            (* split slave state and link state *)
            FOR I := 0 TO MIN(iNumOfSlavesRead, iSLAVEADDR_ARR_SIZE) DO
                (* slave state*)
                arrSlaveInfo[I].stState.eEcState 		:= arrSlaveStates[I].deviceState AND 16#0F;
                arrSlaveInfo[I].stState.bError 			:= arrSlaveStates[I].deviceState.4;
                arrSlaveInfo[I].stState.bInvalidVPRS 	:= arrSlaveStates[I].deviceState.5;
                (* link state *)
                arrSlaveInfo[I].stState.bNoCommToSlave 	:= arrSlaveStates[I].linkState.0;
                arrSlaveInfo[I].stState.bLinkError 		:= arrSlaveStates[I].linkState.1;
                arrSlaveInfo[I].stState.bMissingLink 	:= arrSlaveStates[I].linkState.2;
                arrSlaveInfo[I].stState.bUnexpectedLink := arrSlaveStates[I].linkState.3;
                arrSlaveInfo[I].stState.bPortA 			:= arrSlaveStates[I].linkState.4;
                arrSlaveInfo[I].stState.bPortB 			:= arrSlaveStates[I].linkState.5;
                arrSlaveInfo[I].stState.bPortC 			:= arrSlaveStates[I].linkState.6;
                arrSlaveInfo[I].stState.bPortD 			:= arrSlaveStates[I].linkState.7;
                (* DiagData *)
                arrSlaveInfo[I].bDiagData	:= ((arrSlaveStates[I].deviceState AND 16#F0) <> 0) OR
                    (((arrSlaveStates[I].deviceState AND 16#0F) > 0) AND ((arrSlaveStates[I].deviceState AND 16#0F) < 8)) OR
                    (arrSlaveStates[I].linkState <> 0);

                IF arrSlaveInfo[I].bDiagData THEN
                    IF (I=0) THEN
                        aiDiagIndex[0] := 0;
                    ELSE
                        IF (aiDiagIndex[0] = 0) AND NOT arrSlaveInfo[0].bDiagData THEN
                            aiDiagIndex[0] :=  UDINT_TO_UINT(I);
                        END_IF
                    END_IF
                END_IF
            END_FOR
        END_IF
    END_IF

    IF arrSlaveInfo[aiDiagIndex[0]].bDiagData THEN
        iState := E_EcatDiagState.GetTopoDataLen;
    ELSE
        FOR I := 0 TO ESC_MAX_PORTS DO
            MEMSET(ADR(arrDiagSlaveInfo[I]), 0, SIZEOF(arrDiagSlaveInfo[I]));
            MEMSET(ADR(arrDiagSlaveInfoScanned[I]), 0, SIZEOF(arrDiagSlaveInfoScanned[I]));
        END_FOR
        iState := E_EcatDiagState.Done;
    END_IF
END_IF
END_ACTION

ACTION M_GetTopoData:
fbGetTopologyData(
    NETID	:= sMasterNetID,
    PORT	:= 16#FFFF,
    IDXGRP	:= 16#22,
    IDXOFFS	:= 0,
    LEN		:= iTopologyData*SIZEOF(arrTopologyData[0]),
    DESTADDR:= ADR(arrTopologyData),
    READ	:= TRUE,
    TMOUT	:= tTimeout,
);

IF NOT fbGetTopologyData.BUSY THEN
    fbGetTopologyData(READ := FALSE);

    IF NOT fbGetTopologyData.ERR THEN
        aiDiagPort[0] := arrTopologyData[aiDiagIndex[0]].iOwnPhysicalAddr;
        aiDiagPort[1] := arrTopologyData[aiDiagIndex[0]].stPhysicalAddr.portB;
        aiDiagPort[2] := arrTopologyData[aiDiagIndex[0]].stPhysicalAddr.portC;
        aiDiagPort[ESC_MAX_PORTS] := arrTopologyData[aiDiagIndex[0]].stPhysicalAddr.portD;

        (* clear diag index  *)
        aiDiagIndex[1] := 0;
        aiDiagIndex[2] := 0;
        aiDiagIndex[ESC_MAX_PORTS] := 0;

        (* find slaves on PortB-D of first slave with diag *)
        FOR P := 0 TO ESC_MAX_PORTS DO
            IF aiDiagPort[P] <> 0 THEN
            FOR I := 0 TO MIN(iTopologyData-1,iSLAVEADDR_ARR_SIZE) DO
                IF arrTopologyData[I].iOwnPhysicalAddr = aiDiagPort[P] THEN
                    aiDiagIndex[P] := UDINT_TO_UINT(I);
                    EXIT;
                END_IF
            END_FOR
        END_IF
        END_FOR
    END_IF

    iIdx := 0;
    iState := E_EcatDiagState.ScanSlaves;
END_IF
END_ACTION

ACTION M_GetTopoDataLen:
fbGetTopologyData(
    NETID	:= sMasterNetID,
    PORT	:= 16#FFFF,
    IDXGRP	:= EC_ADS_IGRP_MASTER_COUNT_SLAVE,
    IDXOFFS	:= EC_ADS_IOFFS_MASTER_COUNT_SLAVE,
    LEN		:= SIZEOF(iTopologyData),
    DESTADDR:= ADR(iTopologyData),
    READ	:= TRUE,
    TMOUT	:= tTimeout,
);

IF NOT fbGetTopologyData.BUSY THEN
    fbGetTopologyData(READ := FALSE);

    iState := E_EcatDiagState.GetTopoData;
END_IF
END_ACTION

ACTION M_ScanSlaves:
fbEcGetScannedSlaves(
    bExecute				:= TRUE,
    sNetId					:= sMasterNetID,
    pArrEcScannedSlaveInfo	:= ADR(arrScannedSlaveInfo),
    cbBufLen				:= SIZEOF(arrScannedSlaveInfo),
    tTimeout				:= tTimeout
);

IF NOT fbEcGetScannedSlaves.bBusy THEN
    fbEcGetScannedSlaves(bExecute := FALSE);

    IF fbEcGetScannedSlaves.bError THEN
        nScannedSlaves := 0;
    ELSE
        nScannedSlaves := fbEcGetScannedSlaves.nSlaves;
    END_IF

    iState := E_EcatDiagState.GetSlaveIdentity;

END_IF
END_ACTION

END_FUNCTION_BLOCK

// ---- POUs/Functions/FB_EcatDiag.TcPOU
(*
Ecat bus diagnostic tool
2015-11-4 Alex Wallace
This function block checks the states of all slaves on the ecat bus network,
it could be modified to export the states of the slaves on an individual basis,
but for now it sets the output boolean true if all slaves are OP and false otherwise.
To start the block provide a falling edge on the first pass boolean input.

2018-05-05 Margaret Ghaly
Function block has been modified to retrieve the Device State of the Ethercat Master.
It also exports the states and information of each individual configured Slave.
And saves them in the array q_aEcConfSlaveInfo.
*)
FUNCTION_BLOCK FB_EcatDiag
VAR_INPUT
    {attribute 'naming' := 'omit'}
    I_AMSNetId AT %I* : AMSNETID; //Link to the AMSNETID name in the ethercat master info.
    i_xFirstPass: BOOL; //Hook to system first pass boolean for proper intialization (must be true for the first cycle of the PLC)
END_VAR
VAR_OUTPUT
    q_xAllSlaveStatesGood: BOOL; // Set to True if all Slaves are in OP State
    q_anTermStates: ARRAY[1..256] OF BYTE; //ECAT State of terminals in the bus
    q_xMasterStateGood:BOOL; // Set to True if the Master Device State is OP
    q_nMasterState: WORD; // The Device State of the Master
    q_sMasterState:STRING; //State of the ECAT master
    q_astEcConfSlaveInfo :  ARRAY[1..256] OF ST_EcDevice; //State of all ECAT slaves in the bus
    q_nSlaves: UINT; // the Number of the connected Slaves
END_VAR
VAR
    sNetId: T_AmsNetId; //NetId string
    astTermStates: ARRAY[1..256] OF ST_EcSlaveState; //ECAT Slave States Buffer
    astEcConfSlaveInfo: ARRAY[1..256] OF ST_EcSlaveConfigData; //ECAT Slave Configs Buffer
    fbGetAllSlaveStates: FB_EcGetAllSlaveStates; //Acquires the ECAT Slave States puts them into astTermStates

    fbGetMasterState: FB_EcGetMasterState; //Acquires ECAT Master State
    fbGetConfSlaves: FB_EcGetConfSlaves; //Acquires the ECAT slave configuration of the bus (how many, what kind, etc)
    {attribute 'naming' := 'omit'}
    ftReset: F_TRIG; //Reset trigger sensor
    {attribute 'naming' := 'omit'}
    ftMasterReset: F_TRIG; //Retrigger sensor for GetMasterState
    nIterator: INT; //Generic iterator placeholder
END_VAR

//Create the net ID string
sNetId := F_CreateAmsNetId(I_AMSNetId);

//Query the state of all terminals, collect in astTermStates
ftReset(CLK:=fbGetAllSlaveStates.bBusy OR i_xFirstPass);
fbGetAllSlaveStates.bExecute := ftReset.Q;
fbGetAllSlaveStates(sNetId:=sNetId, pStateBuf := ADR(astTermStates), cbBufLen:=SIZEOF(astTermStates));
//Keep checking...



//Cycle through each entry in the array and check if we have anyone not in OP and that the link state is good.
// If so, then set our global IO bad boolean.
IF fbGetAllSlaveStates.nSlaves > 0 THEN
    q_xAllSlaveStatesGood := TRUE;
FOR nIterator := 1 TO (UINT_TO_INT(fbGetAllSlaveStates.nSlaves) ) BY 1
    DO
    IF NOT( (astTermStates[nIterator].deviceState = EC_DEVICE_STATE_OP) AND (astTermStates[nIterator].linkState = EC_LINK_STATE_OK)) THEN
        q_xAllSlaveStatesGood := FALSE;
    END_IF
    q_anTermStates[nIterator] := astTermStates[nIterator].deviceState;
    q_astEcConfSlaveInfo[nIterator].nDeviceState :=astTermStates[nIterator].deviceState;//
    q_astEcConfSlaveInfo[nIterator].nLinkState :=astTermStates[nIterator].linkState;//
    q_astEcConfSlaveInfo[nIterator].sDeviceState:= F_ConvSlaveStateToString(state:=astTermStates[nIterator]);//

END_FOR
END_IF

// Read the EtherCAT state of the master. If the call is successful,
//the State output variable of type WORD contains the requested status information.
ftMasterReset(CLK:=fbGetMasterState.bBusy OR i_xFirstPass);
fbGetMasterState(sNetId:= sNetId, bExecute:=ftMasterReset.Q,
                state => q_nMasterState,bError=>,
                nErrId=>);
q_xMasterStateGood:= (fbGetMasterState.state = BYTE_TO_UINT(EC_DEVICE_STATE_OP));
q_sMasterState := F_ConvMasterDevStateToString(fbGetMasterState.state);

//This function is used to read a list of all configured slaves from the EtherCat master object Directory
//needs to run only once
fbGetConfSlaves(bExecute := i_xFirstPass, sNetId :=sNetId, pArrEcConfSlaveInfo := ADR(astEcConfSlaveInfo),cbBufLen := SIZEOF(astEcConfSlaveInfo));
q_nSlaves:=fbGetConfSlaves.nSlaves;

IF  NOT (fbGetConfSlaves.bBusy) THEN
    FOR nIterator := 1 TO (UINT_TO_INT(fbGetConfSlaves.nSlaves) ) BY 1
    DO
    q_astEcConfSlaveInfo[nIterator].nAddrr :=astEcConfSlaveInfo[nIterator].nAddr;
    q_astEcConfSlaveInfo[nIterator].sName :=astEcConfSlaveInfo[nIterator].sName;
    q_astEcConfSlaveInfo[nIterator].sType :=astEcConfSlaveInfo[nIterator].sType;
END_FOR
    fbGetConfSlaves.bExecute := FALSE;
END_IF

END_FUNCTION_BLOCK

// ---- POUs/Functions/FB_Index.TcPOU
(* Index FB
A. Wallace 2016-9-3

Why doesn't beckhoff have this as a builtin type?

Use this thing to have a simple indexer with rollover.

*)
FUNCTION_BLOCK FB_Index
VAR_INPUT
    {attribute 'naming' := 'off'}
    LowerLimit : INT := 1; //Incrementer will rollver over to this value (and initialize to this value)
    ValInc : INT := 1; //Incrementer increments by this value
    UpperLimit	:	INT := 1; //Incrementer will rollover at this value to lower limit
    {attribute 'naming' := 'off'}
END_VAR
VAR_OUTPUT

END_VAR
VAR
    nVal	:	INT := LowerLimit; //Internal incrementer value, initialized to LowerLimit
END_VAR

{analysis -2} //Only the methods and actions are needed

ACTION Dec:
nVal := nVal - ValInc;
IF nVal < LowerLimit THEN nVal := UpperLimit; END_IF
END_ACTION

//Decrement the counter and return new value
METHOD DecVal : INT
VAR_INPUT
END_VAR
Dec();
DecVal := nVal;
END_METHOD

ACTION Inc:
// Dont use this, use ValInc
nVal := nVal + ValInc;
IF nVal >  UpperLimit THEN nVal := LowerLimit; END_IF
END_ACTION

//Increment the counter and return new value
METHOD PUBLIC IncVal : INT
VAR_INPUT
END_VAR
Inc();
IncVal := nVal;
END_METHOD

END_FUNCTION_BLOCK

// ---- POUs/Functions/FB_UnixTimeStampGlobal.TcPOU
FUNCTION_BLOCK FB_UnixTimeStampGlobal
(*
    Runs FB_UnixTimeStamp and stuffs the result into this library's GVL
    2019-10-09 Zachary Lentz
*)
VAR_INPUT
    // If TRUE, we will update the output on this cycle.
    bExecute: BOOL;
END_VAR
VAR_OUTPUT
END_VAR
VAR
    fbTimeStamp: FB_UnixTimeStamp;
END_VAR

fbTimeStamp(
    bExecute := bExecute,
    fTime => DefaultGlobals.fTimeStamp);

END_FUNCTION_BLOCK

// ---- POUs/Functions/FB_XKoyoPLCModbus.TcPOU
//Facilitates communication between Beckhoff and Koyo PLC over the network.
FUNCTION_BLOCK FB_XKoyoPLCModbus
VAR
    fbKoyo_PLCInputCoilsRx	:	FB_MBReadCoils; //FB for reading the coils from the other PLC
    anKoyo_PLC_CnBits	:	ARRAY [0..20] OF BYTE; //Buffer for coil readbacks
    {attribute 'naming' := 'omit'}
    ftReset	: F_TRIG; //Reset edge sensor
    {attribute 'naming' := 'omit'}
    tonRetry : TON; //Retry timer
    nIndex : INT; //Index for clearing the coil array
END_VAR

VAR_INPUT
    i_tRetryTime : TIME := T#10S; //Retry time if modbus transaction fails
    i_sIPAddr	 : STRING[15]; //IP address of the Koyo PLC
END_VAR

VAR_OUTPUT
    q_xNoPLCResponse : BOOL := TRUE; //Could not reach the PLC if true
    q_anPLCResponse   : ARRAY [0..20] OF BYTE; //Buffer of coils retrieved from the other PLC
    q_xError         : BOOL := FALSE; //Transaction or other error
END_VAR

(* Look ma' no wires! *)
(* A. Wallace, 2015-7-22
XKoyoPLCModbus

Facilitates communication between Beckhoff and Koyo PLC over the network.

Useful if you don't have time to run a wire. Fairly reliable.

*)

(* Modbus Info for Koyo
Modbus Addresses for
Koyo DL05/06/240/250/260/430/440/450 PLCs
PLC Memory Type		| Modbus start address Decimal (octal) | Function codes
Inputs (X)			  2048 (04000)							2
Special Relays (SP)	  3072 (06000)							2
Outputs (Y)			  2048 (04000)							1, 5, 15
Control Relays (C)	  3072 (06000)							1, 5, 15
Timer Contacts (T)	  6144 (014000)							1, 5, 15
Counter Contacts (CT) 6400 (014400)							1, 5, 15
Stage Status Bits (S) 6144 (012000)							1, 5, 15
*)

(* Begin code *)
// Retry after some time
tonRetry.IN := NOT fbKoyo_PLCInputCoilsRx.bBusy;
tonRetry.PT := i_tRetryTime;
tonRetry();

ftReset(CLK:=fbKoyo_PLCInputCoilsRx.bBusy);
ftReset();

fbKoyo_PLCInputCoilsRx.bExecute := ftReset.Q OR tonRetry.Q;

fbKoyo_PLCInputCoilsRx(sIPAddr:='i_sIPAddr', nTCPPort:=502, nQuantity:=32, nMBAddr:=8#6000, cbLength:=USINT_TO_UDINT(SIZEOF(anKoyo_PLC_CnBits)),  pDestAddr:=ADR(anKoyo_PLC_CnBits), tTimeout:=T#10S);

//run some error code for modbus
IF fbKoyo_PLCInputCoilsRx.bError THEN
    //if there's a modbus error, set all incoming bits to zero
    {analysis -41} //There are one-liners for resetting an array to zero but they don't comply with 61131
    FOR nIndex := 0 TO USINT_TO_INT(SIZEOF(anKoyo_PLC_CnBits))-1 DO //starts at 0
        anKoyo_PLC_CnBits[nIndex]:=0;
    END_FOR
    {analysis +41}
    q_xError := TRUE;

ELSIF ftReset.Q AND fbKoyo_PLCInputCoilsRx.cbRead > 0 THEN
    fbKoyo_PLCInputCoilsRx.bExecute := FALSE;
    q_xNoPLCResponse:= FALSE;
    q_xError := FALSE;

//more error code cause we didn't manage to read anything
ELSIF fbKoyo_PLCInputCoilsRx.cbRead = 0 THEN
    q_xError := TRUE;
    q_xNoPLCResponse:= TRUE;

END_IF

q_anPLCResponse := anKoyo_PLC_CnBits;

END_FUNCTION_BLOCK

// ---- POUs/Hardware/FB_AnalogOutput.TcPOU
FUNCTION_BLOCK FB_AnalogOutput
(*
    Converts a real unit value (e.g., volts) to the integer needed for an analog output terminal.
    2019-10-09 Zachary Lentz
*)
VAR_INPUT
    // The real value to send to the output
    fReal: LREAL;
    // The maximum allowed real value for the connected hardware
    fSafeMax: LREAL;
    // The minimum allowed real value for the connected hardware
    fSafeMin: LREAL;
    // The number of bits correlated with the terminal's max output. This is not necessarily the resolution parameter.
    iTermBits: UINT;
    // The fReal value correlated with the terminal's max output
    fTermMax: LREAL;
    // The fReal value correlated with the terminal's min output
    fTermMin: LREAL;
END_VAR
VAR_OUTPUT
    // Connect this output to the terminal
    iRaw AT %Q*: INT;
END_VAR
VAR
    fScale: LREAL;
END_VAR

// Set the scaling from real to raw
IF fScale = 0 AND fTermMax > fTermMin THEN
    fScale := (EXPT(2, iTermBits) - 1) / (fTermMax - fTermMin);
END_IF

// Adjust real value to be within the limits
fReal := MIN(fReal, fSafeMax, fTermMax);
fReal := MAX(fReal, fSafeMin, fTermMin);

// Scale the output accordingly
iRaw := LREAL_TO_INT((fReal - fTermMin) * fScale);

END_FUNCTION_BLOCK

// ---- POUs/Hardware/FB_AnalogInput.TcPOU
FUNCTION_BLOCK FB_AnalogInput
(*
    Converts the integer from an analog input terminal to a real unit value (e.g., volts)
    2019-10-09 Zachary Lentz
*)
VAR_INPUT
    // Connect this input to the terminal
    iRaw AT %I*: INT;
    // The number of bits correlated with the terminal's max value. This is not necessarily the resolution parameter.
    iTermBits: UINT;
    // The fReal value correlated with the terminal's max value
    fTermMax: LREAL;
    // The fReal value correlated with the terminal's min value
    fTermMin: LREAL;
END_VAR
VAR_OUTPUT
    // The real value read from the output
    fReal: LREAL;
END_VAR
VAR
    fScale: LREAL;
END_VAR

IF fScale = 0 AND fTermMax > fTermMin THEN
    fScale := (EXPT(2, iTermBits) - 1) / (fTermMax - fTermMin);
END_IF
IF fScale <> 0 THEN
    fReal := iRaw / fScale + fTermMin;
END_IF

END_FUNCTION_BLOCK

// ---- POUs/Hardware/FB_CoE_FastRead.TcPOU
FUNCTION_BLOCK FB_CoE_FastRead
(*
    Utility to repeatedly read a CoE parameter
    2019-10-09 Zachary Lentz

    In practice, it's impossible to read most CoE parameters every cycle,
    but this is a best effort and will work if the data is available
*)
VAR_INPUT
    // If TRUE we'll attempt a CoE read this cycle.
    bExecute: BOOL;
    // Link this to your terminal's drive reference variables under InfoData.
    stPlcDriveRef AT %I*: ST_PlcDriveRef;
    // Hexadecimal index of CoE, e.g. the 8010 in 8010:12
    nIndex: UINT;
    // Hexadecimal subindex of CoE, e.g. the 12 in 8010:12
    nSubIndex: BYTE;
    // Pointer to a value to fill with the result of the read, e.g. ADR(MyValue)
    pDstBuf: PVOID;
    // Data size of pDstBuf, e.g. SIZEOF(MyValue)
    cbBufLen: UINT;
END_VAR
VAR_OUTPUT
    // TRUE if the value was updated on this cycle.
    bNewValue: BOOL;
END_VAR
VAR
    fbRead: FB_CoERead_ByDriveRef;
    stDriveRef: ST_DriveRef;
    iLoop: INT;
    bInnerExec: BOOL;
END_VAR

stDriveRef.sNetId := F_CreateAmsNetId(stPlcDriveRef.aNetId);
stDriveRef.nSlaveAddr := stPlcDriveRef.nSlaveAddr;
stDriveRef.nDriveNo := stPlcDriveRef.nDriveNo;
stDriveRef.nDriveType := stPlcDriveRef.nDriveType;

bNewValue := FALSE;
IF bExecute THEN
    // You need to do this block 3 times per cycle to have a chance at always getting a read
    FOR iLoop:= 1 TO 3 DO
        fbRead(
            stDriveRef := stDriveRef,
            nIndex := nIndex,
            nSubIndex := nSubIndex,
            pDstBuf := pDstBuf,
            cbBufLen := cbBufLen,
            bExecute := bInnerExec,
            tTimeout := T#1s);

        IF bInnerExec AND NOT fbRead.bBusy AND NOT fbRead.bError THEN
            bInnerExec := FALSE;
            bNewValue := TRUE;
        ELSE
            bInnerExec := TRUE;
        END_IF
    END_FOR
END_IF

END_FUNCTION_BLOCK

// ---- POUs/Hardware/FB_EL6_Com.TcPOU
FUNCTION_BLOCK FB_EL6_Com
(*
    Communicate with a serial device connected to an EL6XXX
    2019-10-09 Zachary Lentz and Jackson Sheppard

    May contain assumptions about the device we wrote it for, potentially will need to be adjusted
*)
VAR_INPUT
    // Command to send to the serial device
    {attribute 'pytmc' := '
        pv: CMD
        io: io
    '}
    sCmd: STRING;

    // Pulse this to TRUE and back to FALSE when it's time to send
    {attribute 'pytmc' := '
        pv: SEND
        io: io
    '}
    bSend: BOOL;

    // Any static prefix to add before every sent message
    sSendPrefix: STRING;
    // Any static suffix to add after every sent message
    sSendSuffix: STRING;
    // Any static prefix to strip off of every recieved message
    sRecvPrefix: STRING;
    // Any static suffic to strip off of every recieved message
    sRecvSuffix: STRING;
    tTimeout: TIME := T#1S;
END_VAR
VAR_IN_OUT
    stIn_EL6: EL6inData22B;
    stOut_EL6: EL6outData22B;
END_VAR
VAR_OUTPUT
    // The response recieved from the serial device
    {attribute 'pytmc' := '
        pv: RESP
        io: input
    '}
    sResponse: STRING;

    // This is set to TRUE after recieving a response
    {attribute 'pytmc' := '
        pv: DONE
        io: input
    '}
    bDone: BOOL;

    {attribute 'pytmc' := '
        pv: ERR:SER
        io: input
    '}
    eSerialLineErrorID: ComError_t;

    {attribute 'pytmc' := '
        pv: ERR:SEND
        io: input
    '}
    eSendErrorID: ComError_t;

    {attribute 'pytmc' := '
        pv: ERR:RECV
        io: input
    '}
    eRecvErrorID: ComError_t;
END_VAR
VAR
    // Communication Buffers
    TxBuffer: ComBuffer;
    RxBuffer: ComBuffer;
    fbClearComBuffer: ClearComBuffer;

    // Parameters for PLC -> EL6
    fbEL6Ctrl: SerialLineControl;
    bEL6CtrlError: BOOL;
    eEL6CtrlErrorID: ComError_t;

    // Parameters for EL6 -> Serial Device
    fbSend: SendString;
    bSendBusy: BOOL;
    eLastSendErrorID: ComError_t;
    fbReceive: ReceiveString;
    sReceivedString: STRING;
    sLastReceivedString: STRING;
    bStringReceived: BOOL;
    bReceiveBusy: BOOL;
    bReceiveError: BOOL;
    eReceiveErrorID: ComError_t;
    bReceiveTimeout: BOOL;
    nReceiveCounter: UDINT;
    nSendCounter: UDINT;
    sStringToSend: STRING;
    fbFormatString: FB_FormatString;

    // Parameters for state-machine implementation
    nStep: INT := 0;
END_VAR

fbEL6Ctrl(
    Mode:= SERIALLINEMODE_EL6_22B,
    pComIn:= ADR(stIn_EL6),
    pComOut:= ADR(stOut_EL6),
    SizeComIn:= UINT_TO_INT(SIZEOF(stIn_EL6)),
    Error=> ,
    ErrorID=> eSerialLineErrorID,
    TxBuffer:= TxBuffer,
    RxBuffer:= RxBuffer );
IF fbEL6Ctrl.Error THEN
    bEL6CtrlError := TRUE;
    eEL6CtrlErrorID := fbEL6Ctrl.ErrorID;
END_IF
IF bSend THEN
    nStep := 10;
    bSend := FALSE;
    bDone := FALSE;
END_IF
// Attempt at solution that sends one command at a time, not on constant loop
CASE nStep OF
    0:
        ; // idle
    10:
        // Clear buffers in case any lingering data
        fbClearComBuffer(Buffer:=TxBuffer);
        fbClearComBuffer(Buffer:=RxBuffer);
        // Prepare string to send
        sStringToSend := CONCAT(sSendPrefix, CONCAT(sCmd, sSendSuffix));
        // Send string
        fbSend(	SendString:= sStringToSend,
                TXbuffer:= TxBuffer,
                Busy=> bSendBusy,
                Error=> eSendErrorID);
        IF fbSend.Error <> COMERROR_NOERROR THEN
            eLastSendErrorID := fbSend.Error;
        ELSE
            nSendCounter := nSendCounter + 1;
        END_IF
        nStep := nStep + 10;
    20:
        // Finish sending String
        IF fbSend.Busy THEN
            fbSend(	SendString:= sStringToSend,
                    TXbuffer:= TxBuffer,
                    Busy=> bSendBusy,
                    Error=> eSendErrorID);
            IF fbSend.Error <> COMERROR_NOERROR THEN
                eLastSendErrorID := fbSend.Error;
            ELSE
                nSendCounter := nSendCounter + 1;
            END_IF
        ELSE
            nStep := nStep + 10;
        END_IF
    30:
        // Get Reply
        fbReceive(
            Prefix:= sRecvPrefix,
            Suffix:= sRecvSuffix,
            Timeout:= tTimeout,
            ReceivedString:= sReceivedString,
            RXbuffer:= RxBuffer,
            StringReceived=> bStringReceived,
            Busy=> bReceiveBusy,
            Error=> eRecvErrorID,
            RxTimeout=> bReceiveTimeout );
        IF fbReceive.Error <> COMERROR_NOERROR THEN
            eReceiveErrorID := fbReceive.Error;
        END_IF
        IF bStringReceived THEN
            nReceiveCounter := nReceiveCounter + 1;
            // Check for response
            IF FIND(sReceivedString, sStringToSend)=0 THEN
                sResponse := sReceivedString;
                bDone := TRUE;
                nStep := 0;
            END_IF
        END_IF
END_CASE

END_FUNCTION_BLOCK

// ---- POUs/Hardware/FB_LED.TcPOU
FUNCTION_BLOCK FB_LED
(*
    Reads a percentage of illumination determined by the user and converts it to a raw value
    to send to the terminal output via the FB_AnalogOutput.
	
	The determination of the full scale raw value (FSV) is calculated via the iTermBits,
    which is setup as an input variable to be set according to the situation. This value
    is bounded by the FSV of the terminal set by the Beckhoff architecture: (2^15 - 1) = 32767.  
	
	Through the configurable max raw value sent to the terminal output, this LED function block
    is applicable to a wider variety of hardware: whether it be simple Analog Voltage control,
    PWM voltage output, or current controlled output. 

    As an initial application, this FB will be instituted for systems of vaccum chamber LED 
    illuminators on TMO endstations, which are rated for 12 V max. They will be dimmed via the
    EL2502 terminal 24 V PWM output voltage control from 0-50% duty cycle.
	
    2022-5-03 Maarten Thomas-Bosum
*)
VAR_INPUT
	{attribute 'pytmc' := '
        pv: NAME
        io: io 
		field: DESC Descriptive name for the LED
        autosave_pass0: VAL DESC
    '}
	ledName : STRING;
	
	iTermBits : UINT;
	
	{attribute 'pytmc' := '
        pv: ILL:PCT
        field: EGU %
    '}
    fIlluminatorPercent: LREAL;
	
	{attribute 'pytmc' := '
        pv: PWR
        field: ZNAM OFF
        field: ONAM ON
    '}
    bLedPower AT %Q*: BOOL;
END_VAR
VAR
	iIlluminatorINT AT %Q*: INT;
    fbSetIllPercent: FB_AnalogOutput;
END_VAR

// Illuminator conversion to percentage
fbSetIllPercent(
    fReal:=fIlluminatorPercent,
    fSafeMax:=100,
    fSafeMin:=0,
    iTermBits:=iTermBits, 
    fTermMax:=100,
    fTermMin:=0,
    iRaw=>iIlluminatorINT);

IF  fIlluminatorPercent > 0 THEN
	bLedPower := TRUE;
ELSE
	bLEDPower := FALSE;
END_IF

END_FUNCTION_BLOCK

// ---- POUs/Hardware/FB_ThermoCouple.TcPOU
FUNCTION_BLOCK FB_ThermoCouple
(*
    Deprecated as of 2020-03-02, please use FB_TempSensor instead
    2019-10-09 Zachary Lentz
*)
{warning 'Function Block FB_ThermoCouple is deprecated and may be removed in a future release'}
VAR_INPUT
    // Ratio between raw value and actual temperature. Default is 10 for 10 steps per degree (or 0.1 degree resolution)
    iScale: INT := 10;
END_VAR
VAR_OUTPUT
    {attribute 'pytmc' := '
        pv: STC:TEMP
        io: input
    '}
    fTemp: LREAL;

    {attribute 'pytmc' := '
        pv: STC:CONN
        io: input
        field: ONAM Connected
        field: ZNAM Disconnected
    '}
    bConnected: BOOL;

    {attribute 'pytmc' := '
        pv: STC:ERR
        io: input
    '}
    bError AT %I*: BOOL;

    bUnderrange AT %I*: BOOL;
    bOverrange AT %I*: BOOL;
END_VAR
VAR
    iRaw AT %I*: INT;
END_VAR

// The manual states that we are disconnected if we are both overrange and in an error state
bConnected := NOT (bOverrange AND bError);
fTemp := INT_TO_LREAL(iRaw) / iScale;

END_FUNCTION_BLOCK

// ---- POUs/Hardware/FB_TempSensor.TcPOU
FUNCTION_BLOCK FB_TempSensor
(*
    Handles scaling and default diagnostics for temperature sensors,
    such as thermocouples, RTDs, and others.
    2020-03-02 Zachary Lentz
*)
VAR_INPUT
    // Resolution parameter from the Beckhoff docs. Default is 0.1 for 0.1 degree resolution
    fResolution: LREAL := 0.1;
END_VAR
VAR_OUTPUT
    {attribute 'pytmc' := '
        pv: TEMP
        io: input
        field: EGU C
        field: PREC 2
    '}
    fTemp: LREAL;

    {attribute 'pytmc' := '
        pv: CONN
        io: input
        field: ONAM Connected
        field: ZNAM Disconnected
    '}
    bConnected: BOOL;

    {attribute 'pytmc' := '
        pv: ERR
        io: input
        field: ONAM True
        field: ZNAM False
    '}
    bError AT %I*: BOOL := TRUE;

    bUnderrange AT %I*: BOOL;
    bOverrange AT %I*: BOOL;
END_VAR
VAR
    iRaw AT %I*: INT;
END_VAR

// The manual states that we are disconnected if we are both overrange and in an error state
bConnected := NOT (bOverrange AND bError);
fTemp := INT_TO_LREAL(iRaw) * fResolution;

END_FUNCTION_BLOCK

// ---- POUs/Logger/SYSTEM_TIME_TO_RFC3339.TcPOU
//Converts Beckhoff PLC SYSTEMTIME to RFC3339 time format as a string
{attribute 'naming' := 'omit'}
{attribute 'analysis' := '-23'}
FUNCTION SYSTEM_TIME_TO_RFC3339 : STRING(255)
VAR_INPUT
    {attribute 'naming' := 'omit'}
    tCurrentTime	:	TIMESTRUCT; //TIMESTRUCT Time to convert to RFC3339
END_VAR
VAR
END_VAR

SYSTEM_TIME_TO_RFC3339 := CONCAT(REPLACE(SYSTEMTIME_TO_STRING(tCurrentTime), 'T', 1, 11), 'Z');

END_FUNCTION
